(* PLC project STM32 Function Blocks, OpenPLC STM32 Function Blocks Library 1.0, author ERAY YILMAZ *)
(* stored: creationDateTime 2021-11-11T02:33:11, modificationDateTime 2024-06-05T02:33:11 *)

FUNCTION_BLOCK STM32CAN_CONF
  VAR_INPUT
    CONF : BOOL;  (* STM32 CAN Enable pin *)
    BR : LINT;  (* STM32 CAN Baudrate *)
  END_VAR
  VAR_OUTPUT
    DONE : BOOL;  (* STM32 CAN configuration Done flag *)
  END_VAR

END_FUNCTION_BLOCK

FUNCTION_BLOCK STM32CAN_WRITE
  VAR_INPUT
    EN_PIN : BOOL;  (* STM32 CAN Enable pin *)
    CH : USINT;  (* STM32 CAN Channel pin *)
    ID : DWORD;  (* STM32 CAN message ID *)
    D0 : BYTE;  (* STM32 CAN first payload byte *)
    D1 : BYTE;  (* STM32 CAN second payload byte *)
    D2 : BYTE;  (* STM32 CAN third payload byte *)
    D3 : BYTE;  (* STM32 CAN fourth payload byte *)
    D4 : BYTE;  (* STM32 CAN fifth payload byte *)
    D5 : BYTE;  (* STM32 CAN sixth payload byte *)
    D6 : BYTE;  (* STM32 CAN seventh payload byte *)
    D7 : BYTE;  (* STM32 CAN eighth payload byte *)
  END_VAR
  VAR_OUTPUT
    DONE : BOOL;  (* STM32 CAN write done flag *)
  END_VAR

END_FUNCTION_BLOCK

(* CAN READ *)
FUNCTION_BLOCK STM32CAN_READ
  VAR_INPUT
    EN_PIN : BOOL;  (* STM32 CAN Enable pin *)
  END_VAR
  VAR_OUTPUT
    DONE : BOOL;  (* STM32 CAN write done flag *)
    ID : DWORD;  (* STM32 CAN message ID *)
    D0 : BYTE;  (* STM32 CAN first payload byte *)
    D1 : BYTE;  (* STM32 CAN second payload byte *)
    D2 : BYTE;  (* STM32 CAN third payload byte *)
    D3 : BYTE;  (* STM32 CAN fourth payload byte *)
    D4 : BYTE;  (* STM32 CAN fifth payload byte *)
    D5 : BYTE;  (* STM32 CAN sixth payload byte *)
    D6 : BYTE;  (* STM32 CAN seventh payload byte *)
    D7 : BYTE;  (* STM32 CAN eighth payload byte *)
  END_VAR

            DATA := 0;
          
END_FUNCTION_BLOCK
